(* Peeks at the next field tag. This is like calling  "ParseTag", but the
 tag is not consumed. (So a subsequent call to "ParseTag" will return the
same value.)*)
FUNCTION F_PeekTag : HRESULT
VAR_IN_OUT
    stCtx : ST_ParseContext;
END_VAR
VAR_OUTPUT
    nTag : UDINT;
END_VAR

VAR
    nSavedLast : UDINT;
END_VAR

F_PeekTag := S_OK;

IF stCtx.stState.bHasNextTag THEN
    nTag := stCtx.stState.nNextTag;
    RETURN;
END_IF

nSavedLast := stCtx.stState.nLastTag;
F_PeekTag := F_ParseTag(stCtx, nTag=> nTag);
IF FAILED(F_PeekTag) THEN
    RETURN;
END_IF

stCtx.stState.bHasNextTag := TRUE;
stCtx.stState.nNextTag := nTag;
stCtx.stState.nLastTag := nSavedLast; // Undo the side effect of ReadTag

END_FUNCTION

(* stored: Version 1.1.0.1
   POU F_PeekTag: Id {8573c23f-a6ae-4595-a140-59fbe599423b}, SpecialFunc None *)
